INTERFACE I_PtDateTime

END_INTERFACE

(* stored: Version 1.1.0.1, ProductVersion 3.1.4024.12
   Itf I_PtDateTime: Id {63c0eb87-a7d7-4ffe-b48f-2c21ef4e3361} *)
